FUNCTION F_AnyToUnionValue : U_ExpectedOrActual
VAR_INPUT
    AnyValue : ANY;
END_VAR
VAR
    nTempDWORD : DWORD;
    ptREAL : POINTER TO REAL;
    nTempLWORD : LWORD;
    ptLREAL : POINTER TO LREAL;
    ptTIME : POINTER TO TIME;
    ptLTIME : POINTER TO LTIME;

    IteratorCounter : DINT;
    sString : Tc2_System.T_MaxString;
END_VAR

CASE UDINT_TO_INT(AnyValue.TypeClass) OF
    IBaseLibrary.TypeClass.TYPE_BOOL :
        F_AnyToUnionValue.bExpectedOrActual := BYTE_TO_BOOL(AnyValue.pValue[0]);

    IBaseLibrary.TypeClass.TYPE_BIT :
        F_AnyToUnionValue.biExpectedOrActual := BYTE_TO_BIT(AnyValue.pValue[0]);

    IBaseLibrary.TypeClass.TYPE_BYTE :
        F_AnyToUnionValue.nbExpectedOrActual := AnyValue.pValue[0];

    IBaseLibrary.TypeClass.TYPE_WORD :
        F_AnyToUnionValue.nWExpectedOrActual :=
            (SHL(BYTE_TO_WORD(AnyValue.pValue[1]), 8) OR
                 BYTE_TO_WORD(AnyValue.pValue[0]));

    IBaseLibrary.TypeClass.TYPE_DWORD :
        F_AnyToUnionValue.nDWExpectedOrActual :=
            (SHL(SHL(SHL(BYTE_TO_DWORD(AnyValue.pValue[3]), 8) OR
                         BYTE_TO_DWORD(AnyValue.pValue[2]), 8) OR
                         BYTE_TO_DWORD(AnyValue.pValue[1]), 8) OR
                         BYTE_TO_DWORD(AnyValue.pValue[0]));

    IBaseLibrary.TypeClass.TYPE_LWORD :
        F_AnyToUnionValue.nLWExpectedOrActual :=
        (SHL(SHL(SHL(SHL(SHL(SHL(SHL(BYTE_TO_LWORD(AnyValue.pValue[7]), 8) OR
                                     BYTE_TO_LWORD(AnyValue.pValue[6]), 8) OR
                                     BYTE_TO_LWORD(AnyValue.pValue[5]), 8) OR
                                     BYTE_TO_LWORD(AnyValue.pValue[4]), 8) OR
                                     BYTE_TO_LWORD(AnyValue.pValue[3]), 8) OR
                                     BYTE_TO_LWORD(AnyValue.pValue[2]), 8) OR
                                     BYTE_TO_LWORD(AnyValue.pValue[1]), 8) OR
                                     BYTE_TO_LWORD(AnyValue.pValue[0]));

    IBaseLibrary.TypeClass.TYPE_SINT :
        F_AnyToUnionValue.nSExpectedOrActual := BYTE_TO_SINT(AnyValue.pValue[0]);

    IBaseLibrary.TypeClass.TYPE_INT :
        F_AnyToUnionValue.nExpectedOrActual := 
                UINT_TO_INT(SHL(BYTE_TO_UINT(AnyValue.pValue[1]), 8) OR
                                BYTE_TO_UINT(AnyValue.pValue[0]));

    IBaseLibrary.TypeClass.TYPE_DINT :
        F_AnyToUnionValue.nDExpectedOrActual :=
            UDINT_TO_DINT(SHL(SHL(SHL(BYTE_TO_UDINT(AnyValue.pValue[3]), 8) OR
                                      BYTE_TO_UDINT(AnyValue.pValue[2]), 8) OR
                                      BYTE_TO_UDINT(AnyValue.pValue[1]), 8) OR
                                      BYTE_TO_UDINT(AnyValue.pValue[0]));

    IBaseLibrary.TypeClass.TYPE_LINT :
         F_AnyToUnionValue.nLExpectedOrActual :=
        ULINT_TO_LINT(SHL(SHL(SHL(SHL(SHL(SHL(SHL(BYTE_TO_ULINT(AnyValue.pValue[7]), 8) OR
                                                  BYTE_TO_ULINT(AnyValue.pValue[6]), 8) OR
                                                  BYTE_TO_ULINT(AnyValue.pValue[5]), 8) OR
                                                  BYTE_TO_ULINT(AnyValue.pValue[4]), 8) OR
                                                  BYTE_TO_ULINT(AnyValue.pValue[3]), 8) OR
                                                  BYTE_TO_ULINT(AnyValue.pValue[2]), 8) OR
                                                  BYTE_TO_ULINT(AnyValue.pValue[1]), 8) OR
                                                  BYTE_TO_ULINT(AnyValue.pValue[0]));

    IBaseLibrary.TypeClass.TYPE_USINT :
        F_AnyToUnionValue.nUSExpectedOrActual := BYTE_TO_USINT(AnyValue.pValue[0]);

    IBaseLibrary.TypeClass.TYPE_UINT :
        F_AnyToUnionValue.nUExpectedOrActual := 
                (SHL(BYTE_TO_UINT(AnyValue.pValue[1]), 8) OR
                     BYTE_TO_UINT(AnyValue.pValue[0]));

    IBaseLibrary.TypeClass.TYPE_UDINT :
        F_AnyToUnionValue.nUDExpectedOrActual :=
            (SHL(SHL(SHL(BYTE_TO_UDINT(AnyValue.pValue[3]), 8) OR
                         BYTE_TO_UDINT(AnyValue.pValue[2]), 8) OR
                         BYTE_TO_UDINT(AnyValue.pValue[1]), 8) OR
                         BYTE_TO_UDINT(AnyValue.pValue[0]));

    IBaseLibrary.TypeClass.TYPE_ULINT :
        F_AnyToUnionValue.nULExpectedOrActual :=
        (SHL(SHL(SHL(SHL(SHL(SHL(SHL(BYTE_TO_ULINT(AnyValue.pValue[7]), 8) OR
                                     BYTE_TO_ULINT(AnyValue.pValue[6]), 8) OR
                                     BYTE_TO_ULINT(AnyValue.pValue[5]), 8) OR
                                     BYTE_TO_ULINT(AnyValue.pValue[4]), 8) OR
                                     BYTE_TO_ULINT(AnyValue.pValue[3]), 8) OR
                                     BYTE_TO_ULINT(AnyValue.pValue[2]), 8) OR
                                     BYTE_TO_ULINT(AnyValue.pValue[1]), 8) OR
                                     BYTE_TO_ULINT(AnyValue.pValue[0]));

    IBaseLibrary.TypeClass.TYPE_REAL :
        nTempDWORD := (SHL(SHL(SHL(BYTE_TO_DWORD(AnyValue.pValue[3]), 8) OR
                                   BYTE_TO_DWORD(AnyValue.pValue[2]), 8) OR
                                   BYTE_TO_DWORD(AnyValue.pValue[1]), 8) OR
                                   BYTE_TO_DWORD(AnyValue.pValue[0]));
        ptREAL := ADR(nTempDWORD);
        F_AnyToUnionValue.fExpectedOrActual := ptREAL^;

    IBaseLibrary.TypeClass.TYPE_LREAL :
        nTempLWORD := 
        (SHL(SHL(SHL(SHL(SHL(SHL(SHL(BYTE_TO_LWORD(AnyValue.pValue[7]), 8) OR
                                     BYTE_TO_LWORD(AnyValue.pValue[6]), 8) OR
                                     BYTE_TO_LWORD(AnyValue.pValue[5]), 8) OR
                                     BYTE_TO_LWORD(AnyValue.pValue[4]), 8) OR
                                     BYTE_TO_LWORD(AnyValue.pValue[3]), 8) OR
                                     BYTE_TO_LWORD(AnyValue.pValue[2]), 8) OR
                                     BYTE_TO_LWORD(AnyValue.pValue[1]), 8) OR
                                     BYTE_TO_LWORD(AnyValue.pValue[0]));
        ptLREAL := ADR(nTempLWORD);
        F_AnyToUnionValue.fLExpectedOrActual := ptLREAL^;

    IBaseLibrary.TypeClass.TYPE_STRING :
        FOR IteratorCounter := 0 TO MIN(AnyValue.diSize - 1, 254) BY 1 DO
            IF Tc2_System.F_ToCHR(c := AnyValue.pValue[IteratorCounter]) = '$00' THEN
                EXIT;
            END_IF
            sString := Tc2_Standard.CONCAT(STR1 := sString, STR2 := Tc2_System.F_ToCHR(c := AnyValue.pValue[IteratorCounter]));
        END_FOR
        F_AnyToUnionValue.sExpectedOrActual := sString;

    IBaseLibrary.TypeClass.TYPE_WSTRING :
        (* None *)

    IBaseLibrary.TypeClass.TYPE_TIME :
        nTempDWORD := (SHL(SHL(SHL(BYTE_TO_DWORD(AnyValue.pValue[3]), 8) OR
                                   BYTE_TO_DWORD(AnyValue.pValue[2]), 8) OR
                                   BYTE_TO_DWORD(AnyValue.pValue[1]), 8) OR
                                   BYTE_TO_DWORD(AnyValue.pValue[0]));
        ptTIME := ADR(nTempDWORD);
        F_AnyToUnionValue.tExpectedOrActual := ptTIME^;

    IBaseLibrary.TypeClass.TYPE_DATE :
        (* None *)

    IBaseLibrary.TypeClass.TYPE_DATEANDTIME :
        (* None *)

    IBaseLibrary.TypeClass.TYPE_TIMEOFDAY :
        (* None *)

    IBaseLibrary.TypeClass.TYPE_POINTER :
        (* None *)

    IBaseLibrary.TypeClass.TYPE_REFERENCE :
        (* None *)

    IBaseLibrary.TypeClass.TYPE_SUBRANGE :
        (* None *)

    IBaseLibrary.TypeClass.TYPE_ENUM :
        (* None *)

    IBaseLibrary.TypeClass.TYPE_ARRAY :
        (* None *)

    IBaseLibrary.TypeClass.TYPE_PARAMS :
        (* None *)

    IBaseLibrary.TypeClass.TYPE_USERDEF :
        (* None *)

    IBaseLibrary.TypeClass.TYPE_NONE :
        (* None *)

    IBaseLibrary.TypeClass.TYPE_ANY :
        (* None *)

    IBaseLibrary.TypeClass.TYPE_ANYBIT :
        (* None *)

    IBaseLibrary.TypeClass.TYPE_ANYDATE :
        (* None *)

    IBaseLibrary.TypeClass.TYPE_ANYINT :
        (* None *)

    IBaseLibrary.TypeClass.TYPE_ANYNUM :
        (* None *)

    IBaseLibrary.TypeClass.TYPE_ANYREAL :
        (* None *)

    IBaseLibrary.TypeClass.TYPE_LAZY :
        (* None *)

    IBaseLibrary.TypeClass.TYPE_LTIME :
        nTempLWORD := 
        (SHL(SHL(SHL(SHL(SHL(SHL(SHL(BYTE_TO_LWORD(AnyValue.pValue[7]), 8) OR
                                     BYTE_TO_LWORD(AnyValue.pValue[6]), 8) OR
                                     BYTE_TO_LWORD(AnyValue.pValue[5]), 8) OR
                                     BYTE_TO_LWORD(AnyValue.pValue[4]), 8) OR
                                     BYTE_TO_LWORD(AnyValue.pValue[3]), 8) OR
                                     BYTE_TO_LWORD(AnyValue.pValue[2]), 8) OR
                                     BYTE_TO_LWORD(AnyValue.pValue[1]), 8) OR
                                     BYTE_TO_LWORD(AnyValue.pValue[0]));
        ptLTIME := ADR(nTempLWORD);
        F_AnyToUnionValue.ltExpectedOrActual := ptLTIME^;

    IBaseLibrary.TypeClass.TYPE_BITCONST :
        (* None *)

    IBaseLibrary.TypeClass.TYPE_INTERFACE :
        (* None *)

    ELSE
        (* None *)
END_CASE

END_FUNCTION

(* stored: Version 1.1.0.1, ProductVersion 3.1.4022.12
   POU F_AnyToUnionValue: Id {04a97242-7600-4a30-a234-b9e3b1c2770c}, SpecialFunc None *)
